Staubli VAL3: getListPosition.pgx

public program getListPosition(num& x_nIndexX[] (dimensions=1), num& x_nIndexY[] (dimensions=1))
begin
  x_nIndexX=nTopX+1
  x_nIndexY=nFirst+nView+nTopY+1
end
